// TIA Portal V18 export
DATA_BLOCK "FB10-Condition CheckA_DB"   // DB134
VERSION : 0.1
// stored: AutoNumber true, DBAccessibleFromOPCUA true, InstanceOfName FB10-Condition Check, InstanceOfType FB
"FB10-Condition Check"
   // VAR_INPUT
   //    "Time" : DInt;
   //    "Pump ON delay" : DInt;
   //    Check_Time { ExternalAccessible := 'False'; ExternalVisible := 'False'; ExternalWritable := 'False'} : DInt;
   //    Pressure_SP { ExternalAccessible := 'False'; ExternalVisible := 'False'; ExternalWritable := 'False'} : Real;
   //    Pressure_tolerance { ExternalAccessible := 'False'; ExternalVisible := 'False'; ExternalWritable := 'False'} : Real;
   //    Current_pressure { ExternalAccessible := 'False'; ExternalVisible := 'False'; ExternalWritable := 'False'} : Real;
   //    selected { ExternalAccessible := 'False'; ExternalVisible := 'False'; ExternalWritable := 'False'} : Bool;
   // END_VAR
   // VAR_OUTPUT
   //    "dispensing Time PV" : Int;
   //    "Checking Time pv" { ExternalAccessible := 'False'; ExternalVisible := 'False'; ExternalWritable := 'False'} : Int;
   //    test_ok { ExternalAccessible := 'False'; ExternalVisible := 'False'; ExternalWritable := 'False'} : Bool;
   //    test_nok { ExternalAccessible := 'False'; ExternalVisible := 'False'; ExternalWritable := 'False'} : Bool;
   //    test_fail { ExternalAccessible := 'False'; ExternalVisible := 'False'; ExternalWritable := 'False'} : Bool;
   // END_VAR
   // VAR_IN_OUT
   //    "Start ConditonCheck" : Bool;
   //    "Stop ConditonCheck" : Bool;
   //    "ConditonCheck Running" : Bool;
   //    "ConditonCheck completed" : Bool;
   //    "ON Gear Pump" : Bool;
   //    "ON inlet" : Bool;
   // END_VAR
   // VAR
   //    "dispensing time done" : Bool;
   //    "dispensing time in sec" : DInt;
   //    "timer in sec" : DInt;
   //    "timer PV in sec" : DInt;
   //    "timer input" : DInt;
   //    IEC_Timer_0_Instance { S7_SetPoint := 'True'} : TON_TIME;
   //    IEC_Timer_0_Instance_1 { S7_SetPoint := 'True'} : TON_TIME;
   //    IEC_Timer_0_Instance_2 { S7_SetPoint := 'True'} : TON_TIME;
   //    IEC_Timer_0_Instance_4 { S7_SetPoint := 'True'} : TON_TIME;
   //    "Press+ve" { ExternalAccessible := 'False'; ExternalVisible := 'False'; ExternalWritable := 'False'; S7_SetPoint := 'True'} : Real;
   //    "Press-ve" { ExternalAccessible := 'False'; ExternalVisible := 'False'; ExternalWritable := 'False'} : Real;
   //    IEC_Timer_0_Instance_3 { ExternalAccessible := 'False'; ExternalVisible := 'False'; ExternalWritable := 'False'; S7_SetPoint := 'True'} : TON_TIME;
   //    Checktime_ms { ExternalAccessible := 'False'; ExternalVisible := 'False'; ExternalWritable := 'False'; S7_SetPoint := 'True'} : DInt;
   //    Check_timesec { ExternalAccessible := 'False'; ExternalVisible := 'False'; ExternalWritable := 'False'} : DInt;
   //    temp_ons { ExternalAccessible := 'False'; ExternalVisible := 'False'; ExternalWritable := 'False'} : Bool;
   // END_VAR
BEGIN
END_DATA_BLOCK
